// TIA Portal V20 export
FUNCTION_BLOCK "FB_SonplasLoader"   // FB36, SCL
{ S7_Optimized_Access := 'TRUE' }
// stored: MemoryReserve 100, SetENOAutomatically false
   VAR_INPUT
      iOperateInDiagDPCoupler : Bool;
      iOperateInReady : Bool;
      iOperateInNoEStop : Bool;
      iOperateInDoorsClosed : Bool;
      iOperateInRunError : Bool;
      iOperateInOutCollision : Bool;
      iPartInShuttle1Finished : Bool;
      iPartInShuttle2Finished : Bool;
      iPartInDMC_CodeShuttle1 : Array[0..19] of Byte;
      iPartInDMC_CodeShuttle2 : Array[0..19] of Byte;
      "iPartInDMC Code" : Array[0..19] of Byte;
      iMeasureInFlowResultAvail : Bool;
      iMeasureInFlowResult : Int;
      iMeasureInDMC_Code : Array[0..19] of Byte;
   END_VAR
   VAR_OUTPUT
      oOperateOutDiagDPCoupler : Bool;
      oOperateOutReady : Bool;
      oOperateOutNoEStop : Bool;
      oOperateOutDoorsClosed : Bool;
      oOperateOutRunError : Bool;
      oPartOutShuttle1InPos : Bool;
      oPartOutPart1OK : Bool;
      oPartOutPart1NOK : Bool;
      oPartOutShuttle2InPos : Bool;
      oPartOutPart2OK : Bool;
      oPartOutPart2NOK : Bool;
      oPartOutDMC_CodeShuttle1 : Array[0..19] of Byte;
      oPartOutDMC_CodeShuttle2 : Array[0..19] of Byte;
      oPartOutDMC_Code : Array[0..19] of Byte;
      oMeasureOutResultAccepted : Bool;
   END_VAR
   VAR
      sAutomaticMode : Bool;
      sSemiAutoMode : Bool;
      sLastFlowValue : Int;
      sRT_MeasureInFlowResultAvail : R_TRIG;
      sDiagDPCoupler : Bool;
      sReady : Bool;
      sNoEStop : Bool;
      sDoorsClosed : Bool;
      sRunError : Bool;
      sOutCollision : Bool;
      sShuttle1Finished : Bool;
      sShuttle2Finished : Bool;
      sFlowResultAvail : Bool;
      sFlowResult : Real;
      sMeasureDMC_Code : Array[0..19] of Byte;
   END_VAR
   VAR_TEMP
      tIndex : Int;
   END_VAR
BEGIN
   REGION Description header 
       //==================================================================================
       // POSALUX Swiss SA / (C) Copyright 2025
       //----------------------------------------------------------------------------------
       // Title: Initialization of axis
       // Comment/Function: FB_Ext_Loader
       // Author: Fabien WALDT
       // Engineering: TIA Portal v19
       //----------------------------------------------------------------------------------
       // Change log table:
       // Version  | Date     | Expert in charge | Changes applied
       // ---------|----------|------------------|-----------------------------------------
       // 00.00.01 | 20250917 | WFA              | First released version
       // =================================================================================
   END_REGION

   REGION Select automatic / semi automatic mode
       // Keys disabled WFA
       // IF ("LBP_Chan1".E_ProgWait
       //     OR "LBP_Chan1".E_ProgRunning
       //     OR "LBP_Chan1".E_ProgStop)
       //     AND "LBP_ModeGroup".E_AUTO THEN
       //     "DB_McpKeyboardSignals".K10_LoaderAuto.KeyDisable := TRUE;
       //     "DB_McpKeyboardSignals".K11_LoaderSemiAuto.KeyDisable := TRUE;
       //     "DB_HmiKeyboardSignals".K10_LoaderAuto.KeyDisable := TRUE;
       //     "DB_HmiKeyboardSignals".K11_LoaderSemiAuto.KeyDisable := TRUE;
       // ELSE
       //     "DB_McpKeyboardSignals".K10_LoaderAuto.KeyDisable := FALSE;
       //     "DB_McpKeyboardSignals".K11_LoaderSemiAuto.KeyDisable := FALSE;
       //     "DB_HmiKeyboardSignals".K10_LoaderAuto.KeyDisable := FALSE;
       //     "DB_HmiKeyboardSignals".K11_LoaderSemiAuto.KeyDisable := FALSE;
       // END_IF;

       // Mode selection
       #sAutomaticMode := "DB_McpKeyboardSignals".sK10_LoaderAuto.sKeySWToggleStatus;
       // OR "DB_OPC_Machine".State.Current.CurrrentLoadingMode = 1;

       #sSemiAutoMode := "DB_McpKeyboardSignals".sK11_LoaderSemiAuto.sKeySWToggleStatus;
       // OR "DB_OPC_Machine".State.Current.CurrrentLoadingMode = 2;

       // Flip-flop mode selection
       IF "DB_McpKeyboardSignals".sK10_LoaderAuto.sKeySWNegativeFront THEN
           "DB_McpKeyboardSignals".sK11_LoaderSemiAuto.sKeySWToggleStatus := FALSE;
       END_IF;
       IF "DB_McpKeyboardSignals".sK11_LoaderSemiAuto.sKeySWNegativeFront THEN
           "DB_McpKeyboardSignals".sK10_LoaderAuto.sKeySWToggleStatus := FALSE;
       END_IF;

       // LED Management
       "DB_McpKeyboardSignals".sK10_LoaderAuto.sLedSWStatus := "DB_WorkingModes".sAuto;
       "DB_McpKeyboardSignals".sK11_LoaderSemiAuto.sLedSWStatus := "DB_WorkingModes".sSemiAuto;

   END_REGION

   REGION Sonplas Inputs
       REGION Operating_Mode
           // Diagnostic bit DP / DP coupler
           #sDiagDPCoupler := #iOperateInDiagDPCoupler;

           // Sonplas ready
           #sReady := #iOperateInReady;

           // No emergency stop at Sonplas
           #sNoEStop := #iOperateInNoEStop;

           // Safety doors closed at Sonplas
           #sDoorsClosed := #iOperateInDoorsClosed;

           // Running error
           #sRunError := #iOperateInRunError;

           // Loader outside collision area
           #sOutCollision := #iOperateInOutCollision;
       END_REGION

       REGION Part Exchange
           // Posalux Shuttle 1 finished
           #sShuttle1Finished := #iPartInShuttle1Finished;

           // Posalux Shuttle 2 finished
           #sShuttle2Finished := #iPartInShuttle2Finished;
       END_REGION

       REGION Measure
           // Flow result available
           #sFlowResultAvail := #iMeasureInFlowResultAvail;

           // Flow Result
           #sFlowResult := INT_TO_REAL(#iMeasureInFlowResult);

           // Measure DMC Code
           #sMeasureDMC_Code := #iMeasureInDMC_Code;
       END_REGION
   END_REGION

   REGION Measure
       IF #sAutomaticMode OR "DB_WAF".BwLoader.Auto THEN
           #sRT_MeasureInFlowResultAvail(CLK := #sFlowResultAvail);
           IF #sRT_MeasureInFlowResultAvail.Q THEN
               FOR #tIndex := 0 TO 100 DO
                   IF "DB_DataFinalPart".FinalPart[#tIndex].DMC = #"iPartInDMC Code" THEN
                       "DB_DataFinalPart".FinalPart[#tIndex].FlowResult := #sFlowResult;
                       #oMeasureOutResultAccepted := TRUE;
                       EXIT;
                   // ELSE
                       // Product not found WFA A TRAITER
                   END_IF;
               END_FOR;
           ELSIF NOT #iMeasureInFlowResultAvail THEN
               #oMeasureOutResultAccepted := FALSE;
           END_IF;
       ELSE
           #oMeasureOutResultAccepted := FALSE;
       END_IF;
   END_REGION

   REGION Alarmes Messages
       IF "DB_McpKeyboardSignals".sK10_LoaderAuto.sKeySWToggleStatus  AND NOT "DB_LoaderOptions".ExtLoadUnload.Disabled THEN
           // Msg: 700820 "Sonplas - Défaut interface de communication"
           "LBP_AlarmMsgs".UserA[08].A70UUxx[20] := NOT #sDiagDPCoupler;

           // Msg: 700821 "Sonplas - Chargeur pas prêt"
           "LBP_AlarmMsgs".UserA[08].A70UUxx[21] := NOT #sReady;

           // Msg: 700822 "Sonplas - Arrêt d'urgence actif"
           "LBP_AlarmMsgs".UserA[08].A70UUxx[22] := #sNoEStop;

           // Msg: 700823 "Sonplas - Porte(s) ouverte(s)"
           "LBP_AlarmMsgs".UserA[08].A70UUxx[23] := NOT #sDoorsClosed;

           // Msg: 700824 "Sonplas - Running error"
           "LBP_AlarmMsgs".UserA[08].A70UUxx[24] := #sRunError;
       ELSE
           "LBP_AlarmMsgs".UserA[08].A70UUxx[20] := FALSE;
           "LBP_AlarmMsgs".UserA[08].A70UUxx[21] := FALSE;
           "LBP_AlarmMsgs".UserA[08].A70UUxx[22] := FALSE;
           "LBP_AlarmMsgs".UserA[08].A70UUxx[23] := FALSE;
           "LBP_AlarmMsgs".UserA[08].A70UUxx[24] := FALSE;
       END_IF;
   END_REGION

   REGION Sonplas Outputs
       REGION Operating_Mode
           // Diagnostic bit DP / DP coupler
           #oOperateOutDiagDPCoupler := FALSE; // WFA A TRAITER

           // Interface partner ready
           #oOperateOutReady := #sAutomaticMode;

           // No emergency stop at Interface partner
           #oOperateOutNoEStop := NOT "DB_DataFromSafety".EmergencyStop;

           // Safety doors closed at Interface partner
           #oOperateOutDoorsClosed := "DB_DataFromSafety".DoorsClosed;

           // Running error
           #oOperateOutRunError := FALSE; // WFA A TRAITER
       END_REGION

       REGION Part Exchange
           // Shuttle 1 in position
           #oPartOutShuttle1InPos := "DB_LoaderShuttle1".sExtLoadUnload.sCurrent_Step_NB = 40
                                  OR "DB_LoaderShuttle1".sExtLoadUnload.sCurrent_Step_NB = 50
                                  OR "DB_LoaderShuttle1".sExtLoadUnload.sCurrent_Step_NB = 70
                                  OR "DB_LoaderShuttle1".sExtLoadUnload.sCurrent_Step_NB = 80
                                  OR "DB_LoaderShuttle1".sExtLoadUnload.sCurrent_Step_NB = 100
                                  OR "DB_LoaderShuttle1".sExtLoadUnload.sCurrent_Step_NB = 110;

           // Part status 1: OK
           #oPartOutPart1OK := "DB_DataPositions".Position[6].FailCode = 0;

           // Part status 1: nOK
           #oPartOutPart1NOK := "DB_DataPositions".Position[6].FailCode <> 0;

           // Shuttle 2 in position
           #oPartOutShuttle2InPos := "DB_LoaderShuttle2".sExtLoadUnload.sCurrent_Step_NB = 40
                                  OR "DB_LoaderShuttle2".sExtLoadUnload.sCurrent_Step_NB = 50
                                  OR "DB_LoaderShuttle2".sExtLoadUnload.sCurrent_Step_NB = 70
                                  OR "DB_LoaderShuttle2".sExtLoadUnload.sCurrent_Step_NB = 80
                                  OR "DB_LoaderShuttle2".sExtLoadUnload.sCurrent_Step_NB = 100
                                  OR "DB_LoaderShuttle2".sExtLoadUnload.sCurrent_Step_NB = 110;

           // Part status 2: OK
           #oPartOutPart2OK := "DB_DataPositions".Position[7].FailCode = 0;

           // Part status 2: nOK
           #oPartOutPart2NOK := "DB_DataPositions".Position[7].FailCode <> 0;
       END_REGION

       REGION Measure
           // Result accepted
           #oMeasureOutResultAccepted := #oMeasureOutResultAccepted;
       END_REGION
   END_REGION
END_FUNCTION_BLOCK
